(* CoDeSys 2.3.9.50 project: 1B.pr6 *)
(* Libraries: STANDARD.LB6 5.6.98 12:03:02 *)

(* POU MAIN, LD *)
PROGRAM MAIN
VAR
	in1 AT %IX0.0: BOOL;
	in2 AT %IX0.1: BOOL;
	in3 AT %IX0.2: BOOL;
	in4 AT %IX0.3: BOOL;
	redlight AT %QX0.0: BOOL;
	alarm AT %QX0.1: BOOL;
	firedept AT %QX0.2: BOOL;
END_VAR
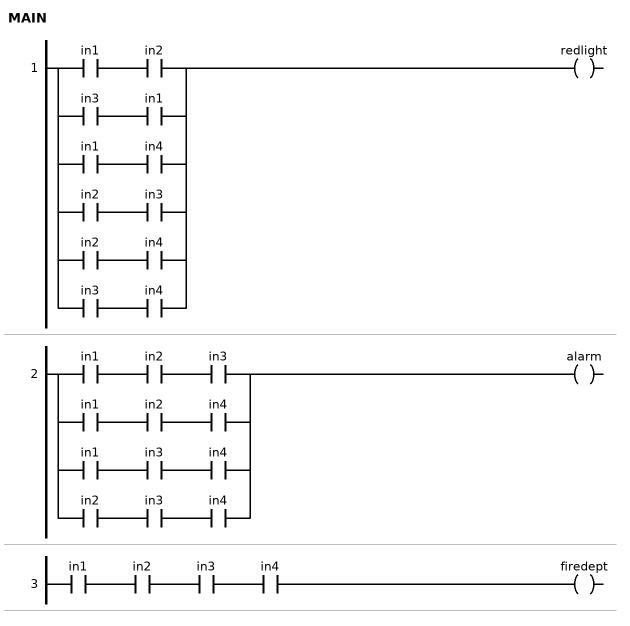
_LD_ (* Ladder Diagram *)
NETWORK 1
	{ [in1] - [in2] | [in3] - [in1] | [in1] - [in4] | [in2] - [in3] | [in2] - [in4] | [in3] - [in4] } --- (redlight)
NETWORK 2
	{ [in1] - [in2] - [in3] | [in1] - [in2] - [in4] | [in1] - [in3] - [in4] | [in2] - [in3] - [in4] } --- (alarm)
NETWORK 3
	[in1] - [in2] - [in3] - [in4] --- (firedept)
_END_LD_
(* the same logic as Structured Text *)
(* Network 1 *)
redlight := in1 AND in2 OR in3 AND in1 OR in1 AND in4 OR in2 AND in3 OR in2 AND in4 OR in3 AND in4;
(* Network 2 *)
alarm := in1 AND in2 AND in3 OR in1 AND in2 AND in4 OR in1 AND in3 AND in4 OR in2 AND in3 AND in4;
(* Network 3 *)
firedept := in1 AND in2 AND in3 AND in4;
END_PROGRAM

(* Visualisation q1Bvisual
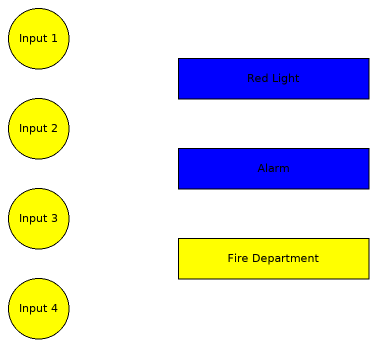
ellipse at (170,180)-(231,241): text "Input 2"; alarm colour if %IX0.1
ellipse at (170,90)-(231,151): text "Input 1"; alarm colour if %IX0.0
ellipse at (170,270)-(231,331): text "Input 3"; alarm colour if %IX0.2
ellipse at (170,360)-(231,421): text "Input 4"; alarm colour if %IX0.3
rectangle at (340,140)-(531,181): text "Red Light"; alarm colour if %QX0.0
rectangle at (340,230)-(531,271): text "Alarm"; alarm colour if %QX0.1
rectangle at (340,320)-(531,361): text "Fire Department"; alarm colour if %QX0.2
*)
